INTERFACE ICyclic EXTENDS __SYSTEM.IQueryInterface

METHOD PUBLIC Cycle : HRESULT
VAR_INPUT
END_VAR
END_METHOD

END_INTERFACE

(* stored: Version 1.1.0.1
   Itf ICyclic: Id {994511c1-43b3-4995-b0c8-49f876ed8799}
   Method Cycle: Id {9328a0f1-a90d-492d-9040-3cf20f5a03ea} *)
